INTERFACE I_VarByteBuffer EXTENDS I_VarByteBufferBase

METHOD Push : BOOL
VAR_INPUT
	pData : pvoid;
	cbSize : UDINT;
END_VAR
END_METHOD

END_INTERFACE

(* stored: Version 1.1.0.1
   Itf I_VarByteBuffer: Id {b8bbd102-587f-43d4-848e-3eac4be39a4b}
   Method Push: Id {b42b1ea6-2cd0-453e-8302-1adb57acab84} *)
